TYPE ST_ZoneRegistryConv :
(**************************************************************************************
 * 	Application		:	BoxControl Framework
 *	Revision		:	$Revision: 404529 $
 *	Revision date	:	$Date: 2018-04-23 08:21:38 +0200 (Mo., 23 Apr 2018) $
 *	Last changed by	:	$Author: b7bolm $
 *	URL				:	$URL: http://almscdc.swisslog.com/repo/SWPD/Development/BoxControlFramework/20_Release/trunk/01_Software/BCF/BCF/JumpStart/20_Product/10_App/10_Base/10_Lib/10_Conv/01_DUTs/ST_ZoneRegistryConv.TcDUT $
 *
 *	Purpose			:	Zone registration structure.
 *
 * ------------------------------------------------------------------------------------
 *	Copyright Swisslog [IP AG], Switzerland. All rights reserved.
 * 
 * ------------------------------------------------------------------------------------
 *	
 * 	Revision History: 
 *
 * 	VERSION			DATE			INITIALS			DESCRIPTION
 *	0.1				01.01.2001		swl					Example
 *
 **************************************************************************************)
STRUCT
	ZoneName			: STRING(System.NAME_LENGTH); // Name as string
	refZoneData			: REFERENCE TO ST_ZoneData; // Internal function data
	refZoneInterface	: REFERENCE TO ST_ZoneInterface; // Function interface data
	HashCode			: UDINT; // HashCode
END_STRUCT
END_TYPE

(* stored: Version 1.1.0.1, ProductVersion 3.1.4022.12
   DUT ST_ZoneRegistryConv: Id {6644bf94-2044-4522-89a8-a6a6c1da8f3d} *)
